FUNCTION_BLOCK FB_OutOnOff
VAR
	//Properties
	bError 				: BOOL 				:= FALSE;

	//value
	bValueOut			: BOOL;

	//Raw value
	bValueInRaw			AT %Q* : BOOL;
END_VAR

PROPERTY Error : BOOL
GET
Error := THIS^.bError;
END_GET
SET
THIS^.bError := Error;
END_SET
END_PROPERTY

PROPERTY ValueOut : BOOL
GET
ValueOut := THIS^.bValueOut;
END_GET
SET
THIS^.bValueOut := ValueOut;
END_SET
END_PROPERTY

METHOD Write
bValueInRaw := bValueOut;
END_METHOD

END_FUNCTION_BLOCK

(* stored: Version 1.1.0.1, ProductVersion 3.1.4024.3
   POU FB_OutOnOff: Id {dba33beb-2add-4d73-999d-97127d9bb5ea}, SpecialFunc None
   Property Error: Id {76fab60f-327b-421a-b545-c3a19badea0c}
   Get Get: Id {4c4480c7-9d76-4089-8899-453ac209bb8c}
   Set Set: Id {0ce510f0-717e-499e-8907-cafdf3228545}
   Property ValueOut: Id {4e245188-4580-44db-b5aa-be6d9c44162b}
   Get Get: Id {fdb7fb88-dd91-4958-9fc9-2d8c6551dbbb}
   Set Set: Id {56dd7628-9ab1-48fe-9b6c-93a8fdabf7bb}
   Method Write: Id {ddc78650-7f0a-4902-bc34-3aeeb4b8017a} *)
